PROGRAM P5_04_BatchStatus
VAR
	tonBatchOpen			:TON;
	tPhaseTimeET			:TIME;
	tSubStep1Prod			:TIME;
	tSubStep1				:TIME;
	tSubStep2				:TIME;
	tSubStep3				:TIME;
	tSubStep4				:TIME;
	tSubStep5				:TIME;
	tSubStep6				:TIME;
	tSubStep7				:TIME;
	
	tSubStep1pt				:TIME;
	tSubStep2pt				:TIME;
	tSubStep3pt				:TIME;
	tSubStep4pt				:TIME;
	tSubStep5pt				:TIME;
	tSubStep6pt				:TIME;
	tSubStep7pt				:TIME;
	
	
	bHoldBar1				:BOOL;
	bHoldBar2				:BOOL;
	bHoldBar3				:BOOL;
	bHoldBar4				:BOOL;
	bHoldBar5				:BOOL;
	bHoldBar6				:BOOL;
	bHoldBar7				:BOOL;
	
	
	iCurrProc				:INT;
	

END_VAR
VAR // added by the converter: edge detectors and wires of the graphical bodies
    _w1, _w2, _w3, _w4, _w5, _w6, _w7, _w8, _w9, _w10, _w11, _w12, _w13, _w14, _w15 : TIME;
    _w16 : BOOL;
END_VAR

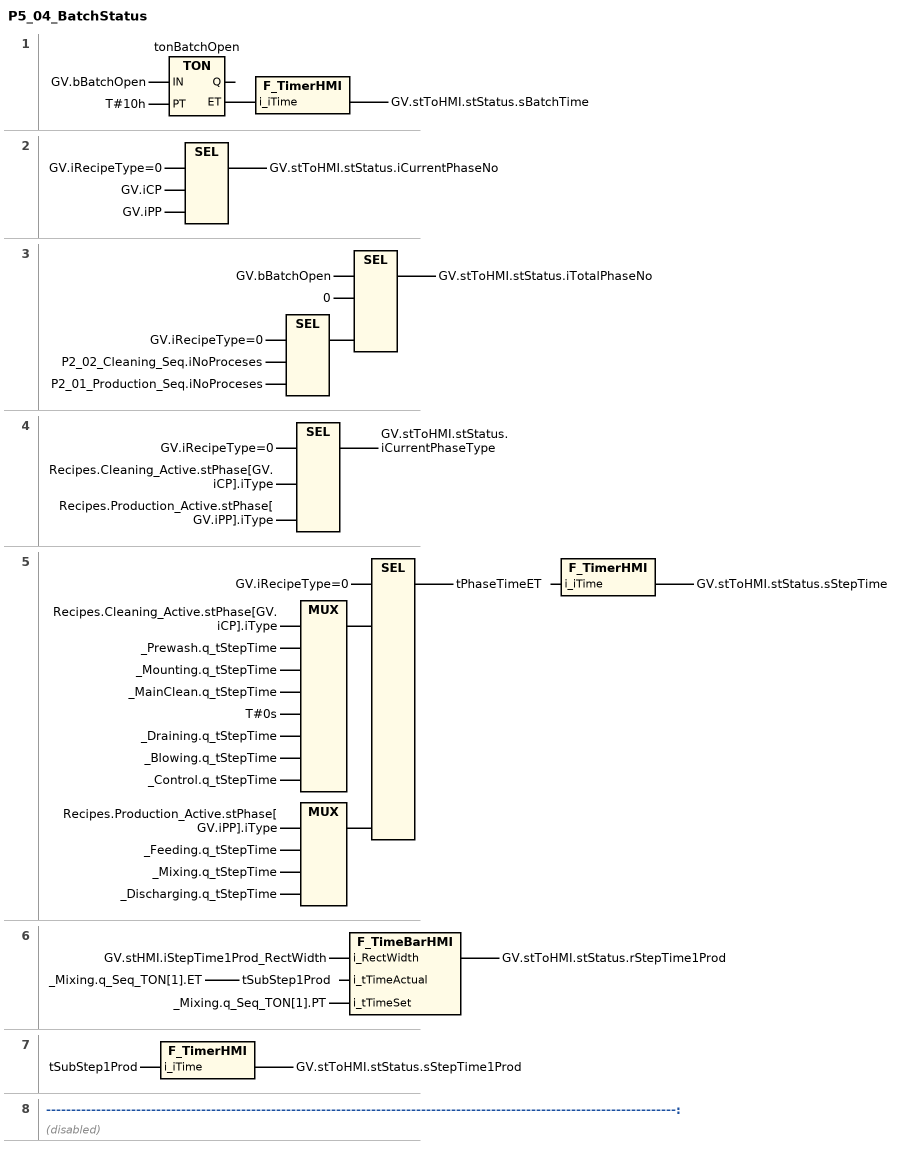
// NETWORK 1
tonBatchOpen(IN := GV.bBatchOpen, PT := T#10h); // TON
GV.stToHMI.stStatus.sBatchTime := F_TimerHMI(i_iTime := tonBatchOpen.ET);

// NETWORK 2
GV.stToHMI.stStatus.iCurrentPhaseNo := SEL(GV.iRecipeType=0, GV.iCP, GV.iPP);

// NETWORK 3
GV.stToHMI.stStatus.iTotalPhaseNo := SEL(GV.bBatchOpen, 0, SEL(GV.iRecipeType=0, P2_02_Cleaning_Seq.iNoProceses, P2_01_Production_Seq.iNoProceses));

// NETWORK 4
GV.stToHMI.stStatus.iCurrentPhaseType := SEL(GV.iRecipeType=0, Recipes.Cleaning_Active.stPhase[GV.iCP].iType, Recipes.Production_Active.stPhase[GV.iPP].iType);

// NETWORK 5
_w1 := SEL(GV.iRecipeType=0, MUX(Recipes.Cleaning_Active.stPhase[GV.iCP].iType, _Prewash.q_tStepTime, _Mounting.q_tStepTime, _MainClean.q_tStepTime, T#0s, _Draining.q_tStepTime, _Blowing.q_tStepTime, _Control.q_tStepTime), MUX(Recipes.Production_Active.stPhase[GV.iPP].iType, _Feeding.q_tStepTime, _Mixing.q_tStepTime, _Discharging.q_tStepTime));
tPhaseTimeET := _w1;
GV.stToHMI.stStatus.sStepTime := F_TimerHMI(i_iTime := _w1);

// NETWORK 6
tSubStep1Prod := _Mixing.q_Seq_TON[1].ET;
GV.stToHMI.stStatus.rStepTime1Prod := F_TimeBarHMI(i_RectWidth := GV.stHMI.iStepTime1Prod_RectWidth, i_tTimeActual := _Mixing.q_Seq_TON[1].ET, i_tTimeSet := _Mixing.q_Seq_TON[1].PT);

// NETWORK 7
GV.stToHMI.stStatus.sStepTime1Prod := F_TimerHMI(i_iTime := tSubStep1Prod);

// NETWORK 8 (disabled)
// label: ------------------------------------------------------------------------------------------------------------------------------

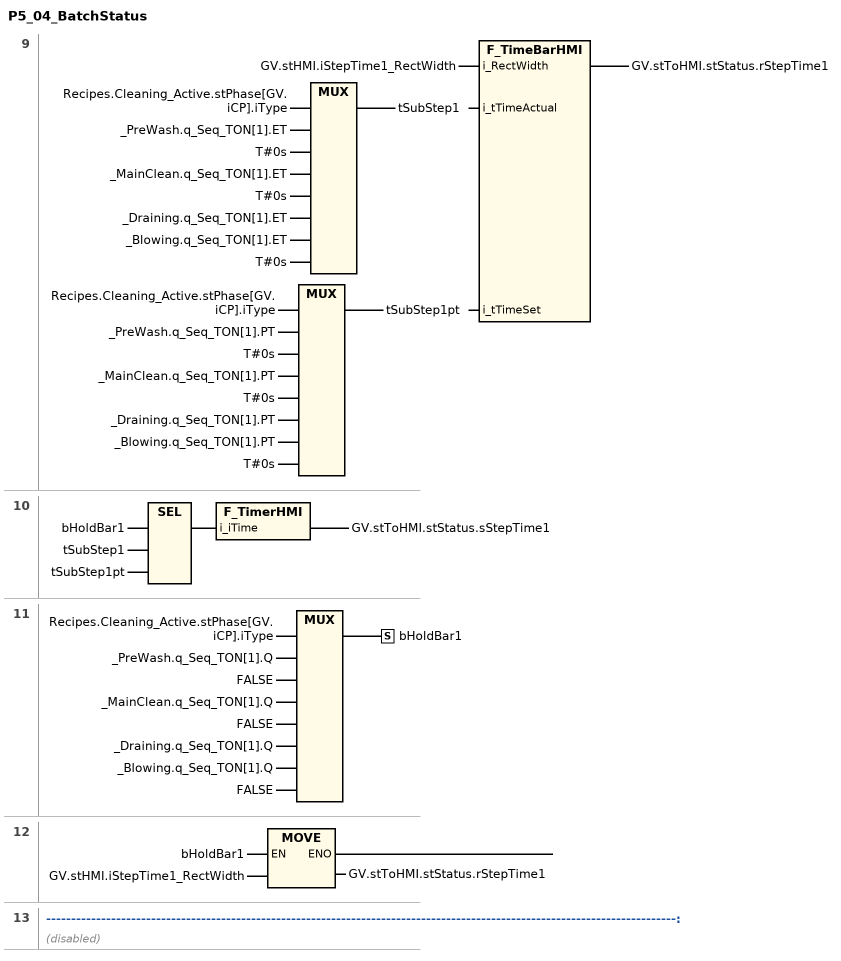
// NETWORK 9
_w2 := MUX(Recipes.Cleaning_Active.stPhase[GV.iCP].iType, _PreWash.q_Seq_TON[1].ET, T#0s, _MainClean.q_Seq_TON[1].ET, T#0s, _Draining.q_Seq_TON[1].ET, _Blowing.q_Seq_TON[1].ET, T#0s);
tSubStep1 := _w2;
_w3 := MUX(Recipes.Cleaning_Active.stPhase[GV.iCP].iType, _PreWash.q_Seq_TON[1].PT, T#0s, _MainClean.q_Seq_TON[1].PT, T#0s, _Draining.q_Seq_TON[1].PT, _Blowing.q_Seq_TON[1].PT, T#0s);
tSubStep1pt := _w3;
GV.stToHMI.stStatus.rStepTime1 := F_TimeBarHMI(i_RectWidth := GV.stHMI.iStepTime1_RectWidth, i_tTimeActual := _w2, i_tTimeSet := _w3);

// NETWORK 10
GV.stToHMI.stStatus.sStepTime1 := F_TimerHMI(i_iTime := SEL(bHoldBar1, tSubStep1, tSubStep1pt));

// NETWORK 11
bHoldBar1 S= MUX(Recipes.Cleaning_Active.stPhase[GV.iCP].iType, _PreWash.q_Seq_TON[1].Q, FALSE, _MainClean.q_Seq_TON[1].Q, FALSE, _Draining.q_Seq_TON[1].Q, _Blowing.q_Seq_TON[1].Q, FALSE);

// NETWORK 12
IF bHoldBar1 THEN GV.stToHMI.stStatus.rStepTime1 := GV.stHMI.iStepTime1_RectWidth; END_IF

// NETWORK 13 (disabled)
// label: ------------------------------------------------------------------------------------------------------------------------------

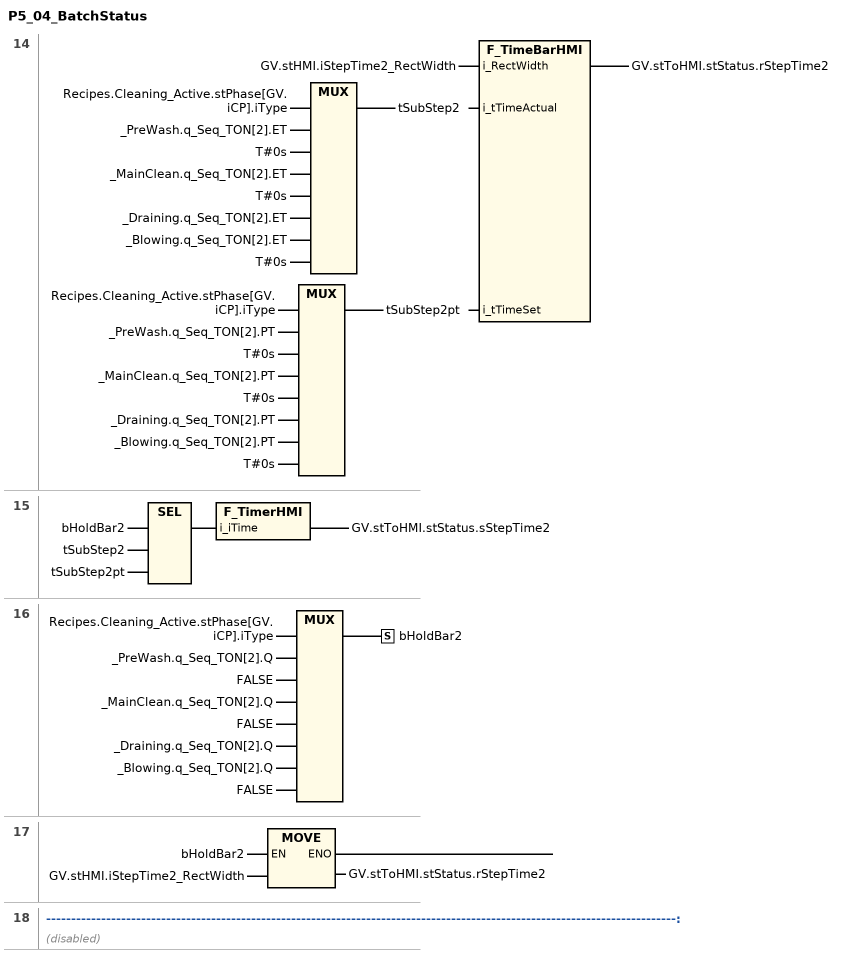
// NETWORK 14
_w4 := MUX(Recipes.Cleaning_Active.stPhase[GV.iCP].iType, _PreWash.q_Seq_TON[2].ET, T#0s, _MainClean.q_Seq_TON[2].ET, T#0s, _Draining.q_Seq_TON[2].ET, _Blowing.q_Seq_TON[2].ET, T#0s);
tSubStep2 := _w4;
_w5 := MUX(Recipes.Cleaning_Active.stPhase[GV.iCP].iType, _PreWash.q_Seq_TON[2].PT, T#0s, _MainClean.q_Seq_TON[2].PT, T#0s, _Draining.q_Seq_TON[2].PT, _Blowing.q_Seq_TON[2].PT, T#0s);
tSubStep2pt := _w5;
GV.stToHMI.stStatus.rStepTime2 := F_TimeBarHMI(i_RectWidth := GV.stHMI.iStepTime2_RectWidth, i_tTimeActual := _w4, i_tTimeSet := _w5);

// NETWORK 15
GV.stToHMI.stStatus.sStepTime2 := F_TimerHMI(i_iTime := SEL(bHoldBar2, tSubStep2, tSubStep2pt));

// NETWORK 16
bHoldBar2 S= MUX(Recipes.Cleaning_Active.stPhase[GV.iCP].iType, _PreWash.q_Seq_TON[2].Q, FALSE, _MainClean.q_Seq_TON[2].Q, FALSE, _Draining.q_Seq_TON[2].Q, _Blowing.q_Seq_TON[2].Q, FALSE);

// NETWORK 17
IF bHoldBar2 THEN GV.stToHMI.stStatus.rStepTime2 := GV.stHMI.iStepTime2_RectWidth; END_IF

// NETWORK 18 (disabled)
// label: ------------------------------------------------------------------------------------------------------------------------------

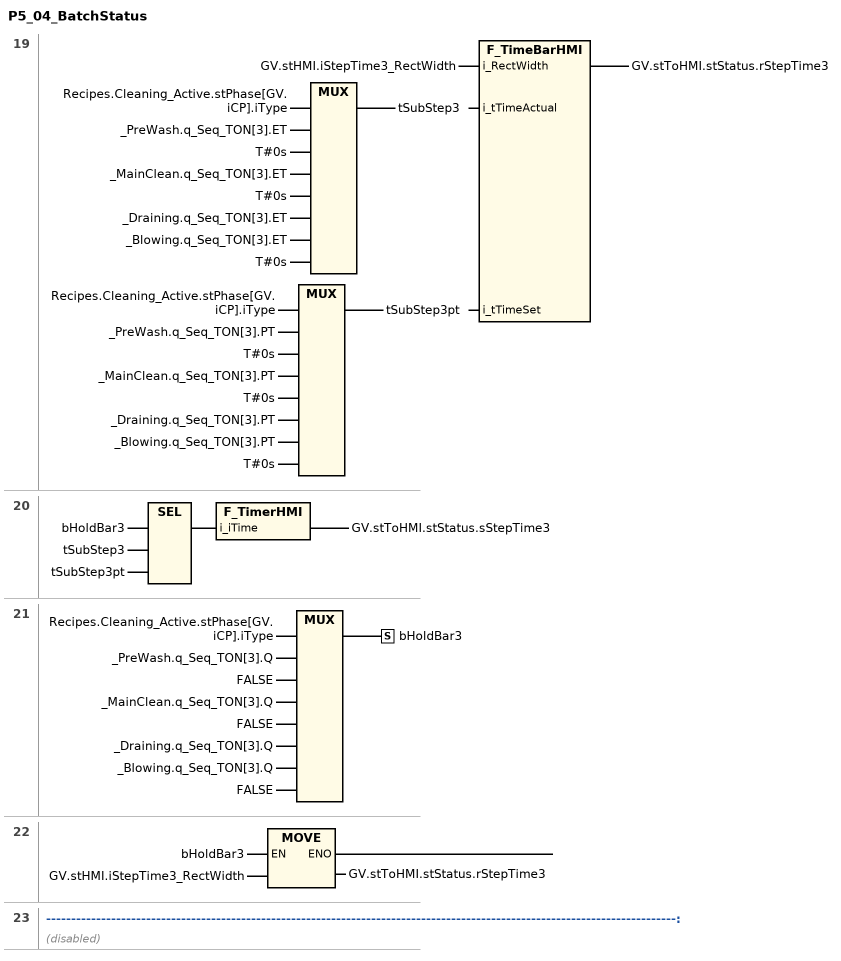
// NETWORK 19
_w6 := MUX(Recipes.Cleaning_Active.stPhase[GV.iCP].iType, _PreWash.q_Seq_TON[3].ET, T#0s, _MainClean.q_Seq_TON[3].ET, T#0s, _Draining.q_Seq_TON[3].ET, _Blowing.q_Seq_TON[3].ET, T#0s);
tSubStep3 := _w6;
_w7 := MUX(Recipes.Cleaning_Active.stPhase[GV.iCP].iType, _PreWash.q_Seq_TON[3].PT, T#0s, _MainClean.q_Seq_TON[3].PT, T#0s, _Draining.q_Seq_TON[3].PT, _Blowing.q_Seq_TON[3].PT, T#0s);
tSubStep3pt := _w7;
GV.stToHMI.stStatus.rStepTime3 := F_TimeBarHMI(i_RectWidth := GV.stHMI.iStepTime3_RectWidth, i_tTimeActual := _w6, i_tTimeSet := _w7);

// NETWORK 20
GV.stToHMI.stStatus.sStepTime3 := F_TimerHMI(i_iTime := SEL(bHoldBar3, tSubStep3, tSubStep3pt));

// NETWORK 21
bHoldBar3 S= MUX(Recipes.Cleaning_Active.stPhase[GV.iCP].iType, _PreWash.q_Seq_TON[3].Q, FALSE, _MainClean.q_Seq_TON[3].Q, FALSE, _Draining.q_Seq_TON[3].Q, _Blowing.q_Seq_TON[3].Q, FALSE);

// NETWORK 22
IF bHoldBar3 THEN GV.stToHMI.stStatus.rStepTime3 := GV.stHMI.iStepTime3_RectWidth; END_IF

// NETWORK 23 (disabled)
// label: ------------------------------------------------------------------------------------------------------------------------------

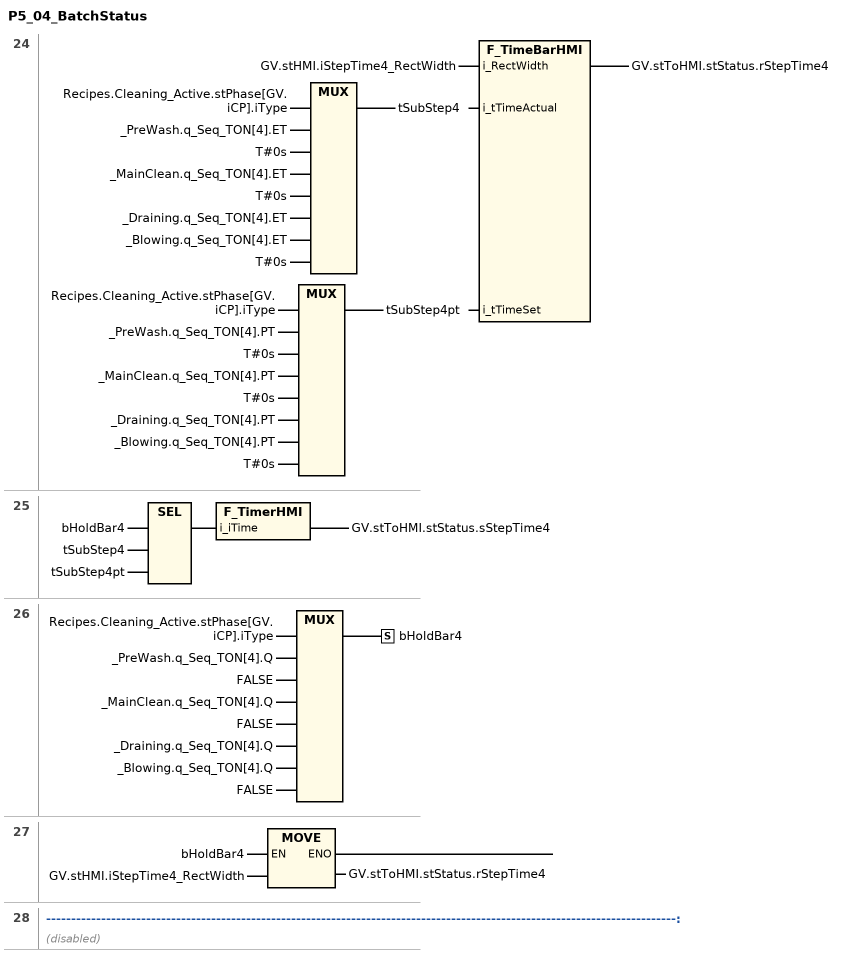
// NETWORK 24
_w8 := MUX(Recipes.Cleaning_Active.stPhase[GV.iCP].iType, _PreWash.q_Seq_TON[4].ET, T#0s, _MainClean.q_Seq_TON[4].ET, T#0s, _Draining.q_Seq_TON[4].ET, _Blowing.q_Seq_TON[4].ET, T#0s);
tSubStep4 := _w8;
_w9 := MUX(Recipes.Cleaning_Active.stPhase[GV.iCP].iType, _PreWash.q_Seq_TON[4].PT, T#0s, _MainClean.q_Seq_TON[4].PT, T#0s, _Draining.q_Seq_TON[4].PT, _Blowing.q_Seq_TON[4].PT, T#0s);
tSubStep4pt := _w9;
GV.stToHMI.stStatus.rStepTime4 := F_TimeBarHMI(i_RectWidth := GV.stHMI.iStepTime4_RectWidth, i_tTimeActual := _w8, i_tTimeSet := _w9);

// NETWORK 25
GV.stToHMI.stStatus.sStepTime4 := F_TimerHMI(i_iTime := SEL(bHoldBar4, tSubStep4, tSubStep4pt));

// NETWORK 26
bHoldBar4 S= MUX(Recipes.Cleaning_Active.stPhase[GV.iCP].iType, _PreWash.q_Seq_TON[4].Q, FALSE, _MainClean.q_Seq_TON[4].Q, FALSE, _Draining.q_Seq_TON[4].Q, _Blowing.q_Seq_TON[4].Q, FALSE);

// NETWORK 27
IF bHoldBar4 THEN GV.stToHMI.stStatus.rStepTime4 := GV.stHMI.iStepTime4_RectWidth; END_IF

// NETWORK 28 (disabled)
// label: ------------------------------------------------------------------------------------------------------------------------------

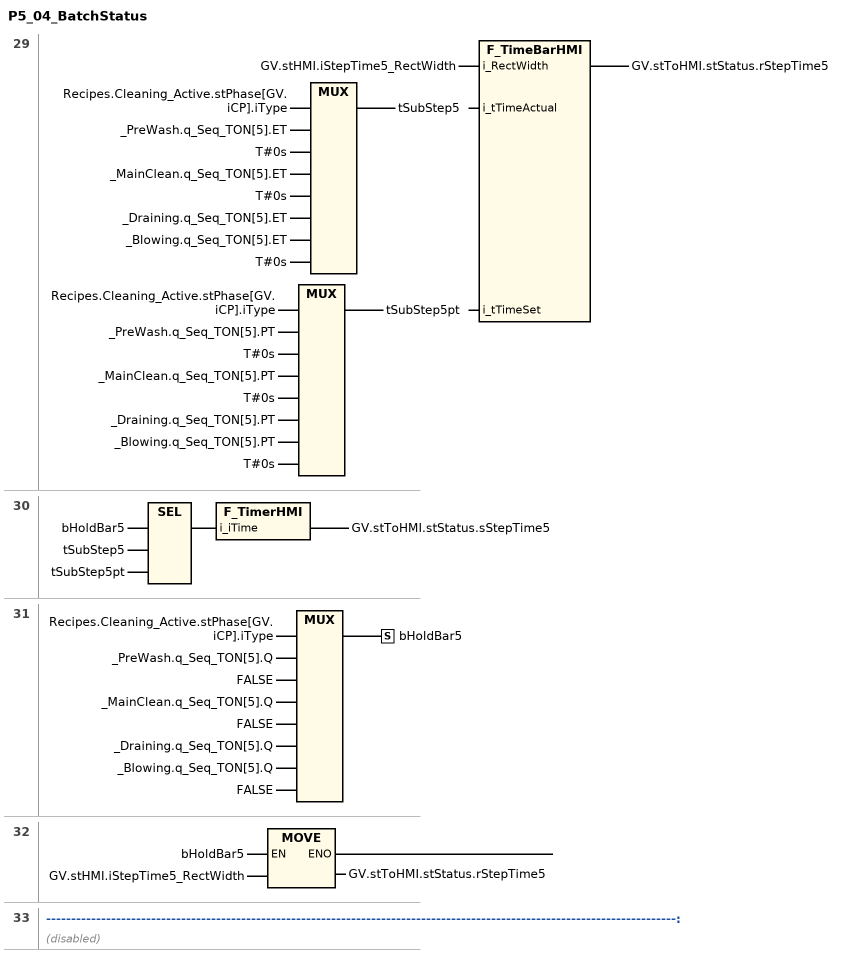
// NETWORK 29
_w10 := MUX(Recipes.Cleaning_Active.stPhase[GV.iCP].iType, _PreWash.q_Seq_TON[5].ET, T#0s, _MainClean.q_Seq_TON[5].ET, T#0s, _Draining.q_Seq_TON[5].ET, _Blowing.q_Seq_TON[5].ET, T#0s);
tSubStep5 := _w10;
_w11 := MUX(Recipes.Cleaning_Active.stPhase[GV.iCP].iType, _PreWash.q_Seq_TON[5].PT, T#0s, _MainClean.q_Seq_TON[5].PT, T#0s, _Draining.q_Seq_TON[5].PT, _Blowing.q_Seq_TON[5].PT, T#0s);
tSubStep5pt := _w11;
GV.stToHMI.stStatus.rStepTime5 := F_TimeBarHMI(i_RectWidth := GV.stHMI.iStepTime5_RectWidth, i_tTimeActual := _w10, i_tTimeSet := _w11);

// NETWORK 30
GV.stToHMI.stStatus.sStepTime5 := F_TimerHMI(i_iTime := SEL(bHoldBar5, tSubStep5, tSubStep5pt));

// NETWORK 31
bHoldBar5 S= MUX(Recipes.Cleaning_Active.stPhase[GV.iCP].iType, _PreWash.q_Seq_TON[5].Q, FALSE, _MainClean.q_Seq_TON[5].Q, FALSE, _Draining.q_Seq_TON[5].Q, _Blowing.q_Seq_TON[5].Q, FALSE);

// NETWORK 32
IF bHoldBar5 THEN GV.stToHMI.stStatus.rStepTime5 := GV.stHMI.iStepTime5_RectWidth; END_IF

// NETWORK 33 (disabled)
// label: ------------------------------------------------------------------------------------------------------------------------------

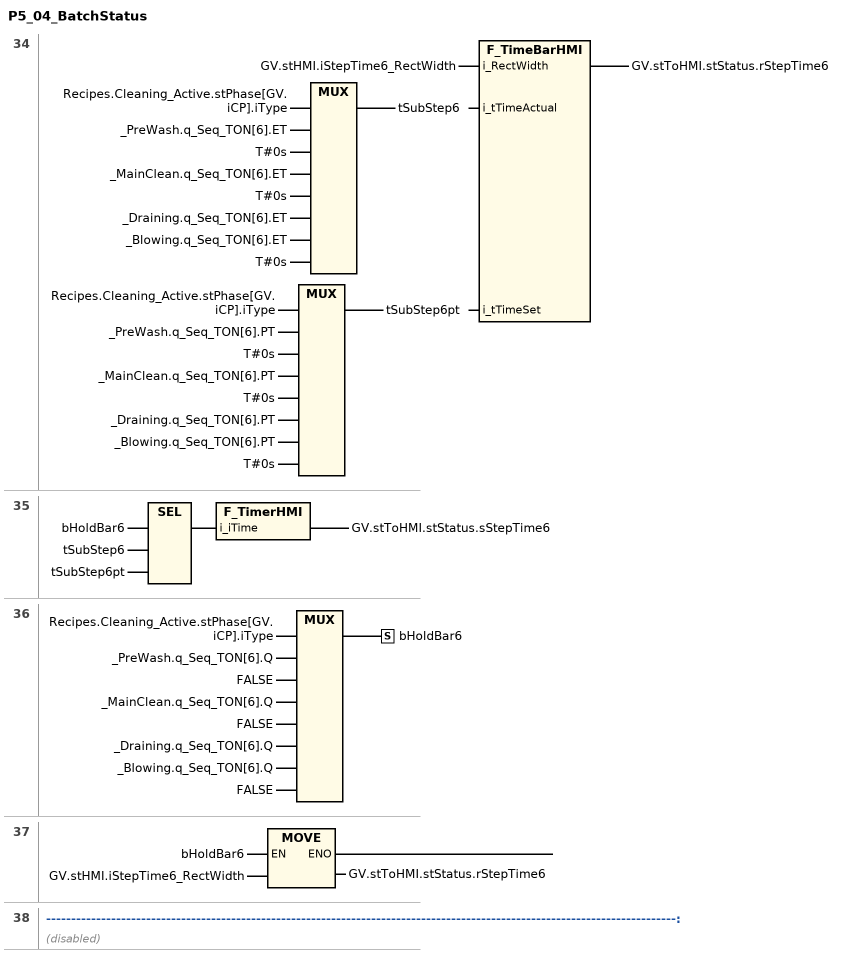
// NETWORK 34
_w12 := MUX(Recipes.Cleaning_Active.stPhase[GV.iCP].iType, _PreWash.q_Seq_TON[6].ET, T#0s, _MainClean.q_Seq_TON[6].ET, T#0s, _Draining.q_Seq_TON[6].ET, _Blowing.q_Seq_TON[6].ET, T#0s);
tSubStep6 := _w12;
_w13 := MUX(Recipes.Cleaning_Active.stPhase[GV.iCP].iType, _PreWash.q_Seq_TON[6].PT, T#0s, _MainClean.q_Seq_TON[6].PT, T#0s, _Draining.q_Seq_TON[6].PT, _Blowing.q_Seq_TON[6].PT, T#0s);
tSubStep6pt := _w13;
GV.stToHMI.stStatus.rStepTime6 := F_TimeBarHMI(i_RectWidth := GV.stHMI.iStepTime6_RectWidth, i_tTimeActual := _w12, i_tTimeSet := _w13);

// NETWORK 35
GV.stToHMI.stStatus.sStepTime6 := F_TimerHMI(i_iTime := SEL(bHoldBar6, tSubStep6, tSubStep6pt));

// NETWORK 36
bHoldBar6 S= MUX(Recipes.Cleaning_Active.stPhase[GV.iCP].iType, _PreWash.q_Seq_TON[6].Q, FALSE, _MainClean.q_Seq_TON[6].Q, FALSE, _Draining.q_Seq_TON[6].Q, _Blowing.q_Seq_TON[6].Q, FALSE);

// NETWORK 37
IF bHoldBar6 THEN GV.stToHMI.stStatus.rStepTime6 := GV.stHMI.iStepTime6_RectWidth; END_IF

// NETWORK 38 (disabled)
// label: ------------------------------------------------------------------------------------------------------------------------------

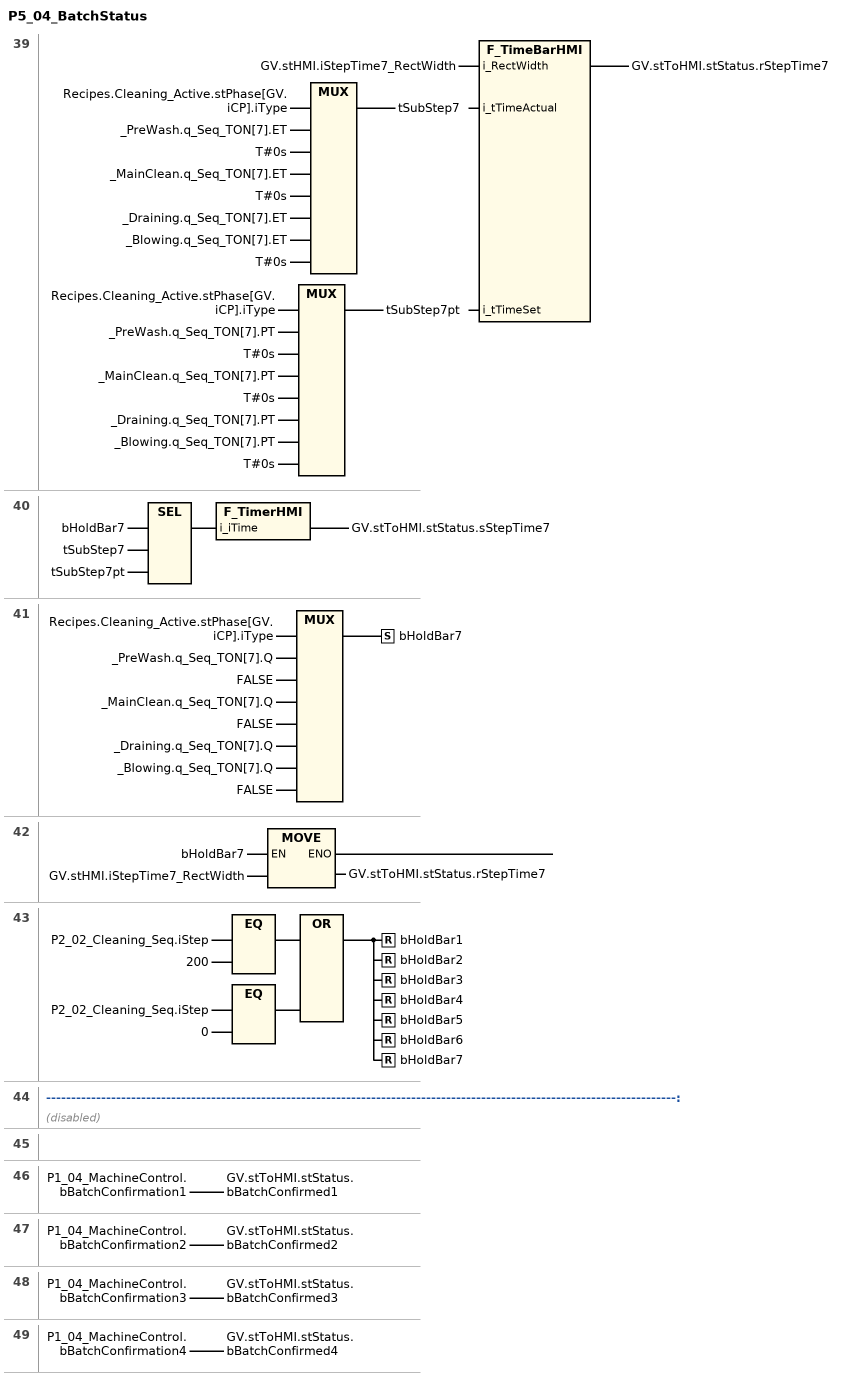
// NETWORK 39
_w14 := MUX(Recipes.Cleaning_Active.stPhase[GV.iCP].iType, _PreWash.q_Seq_TON[7].ET, T#0s, _MainClean.q_Seq_TON[7].ET, T#0s, _Draining.q_Seq_TON[7].ET, _Blowing.q_Seq_TON[7].ET, T#0s);
tSubStep7 := _w14;
_w15 := MUX(Recipes.Cleaning_Active.stPhase[GV.iCP].iType, _PreWash.q_Seq_TON[7].PT, T#0s, _MainClean.q_Seq_TON[7].PT, T#0s, _Draining.q_Seq_TON[7].PT, _Blowing.q_Seq_TON[7].PT, T#0s);
tSubStep7pt := _w15;
GV.stToHMI.stStatus.rStepTime7 := F_TimeBarHMI(i_RectWidth := GV.stHMI.iStepTime7_RectWidth, i_tTimeActual := _w14, i_tTimeSet := _w15);

// NETWORK 40
GV.stToHMI.stStatus.sStepTime7 := F_TimerHMI(i_iTime := SEL(bHoldBar7, tSubStep7, tSubStep7pt));

// NETWORK 41
bHoldBar7 S= MUX(Recipes.Cleaning_Active.stPhase[GV.iCP].iType, _PreWash.q_Seq_TON[7].Q, FALSE, _MainClean.q_Seq_TON[7].Q, FALSE, _Draining.q_Seq_TON[7].Q, _Blowing.q_Seq_TON[7].Q, FALSE);

// NETWORK 42
IF bHoldBar7 THEN GV.stToHMI.stStatus.rStepTime7 := GV.stHMI.iStepTime7_RectWidth; END_IF

// NETWORK 43
_w16 := P2_02_Cleaning_Seq.iStep = 200 OR P2_02_Cleaning_Seq.iStep = 0;
bHoldBar1 R= _w16;
bHoldBar2 R= _w16;
bHoldBar3 R= _w16;
bHoldBar4 R= _w16;
bHoldBar5 R= _w16;
bHoldBar6 R= _w16;
bHoldBar7 R= _w16;

// NETWORK 44 (disabled)
// label: ------------------------------------------------------------------------------------------------------------------------------

// NETWORK 45

// NETWORK 46
GV.stToHMI.stStatus.bBatchConfirmed1 := P1_04_MachineControl.bBatchConfirmation1;

// NETWORK 47
GV.stToHMI.stStatus.bBatchConfirmed2 := P1_04_MachineControl.bBatchConfirmation2;

// NETWORK 48
GV.stToHMI.stStatus.bBatchConfirmed3 := P1_04_MachineControl.bBatchConfirmation3;

// NETWORK 49
GV.stToHMI.stStatus.bBatchConfirmed4 := P1_04_MachineControl.bBatchConfirmation4;

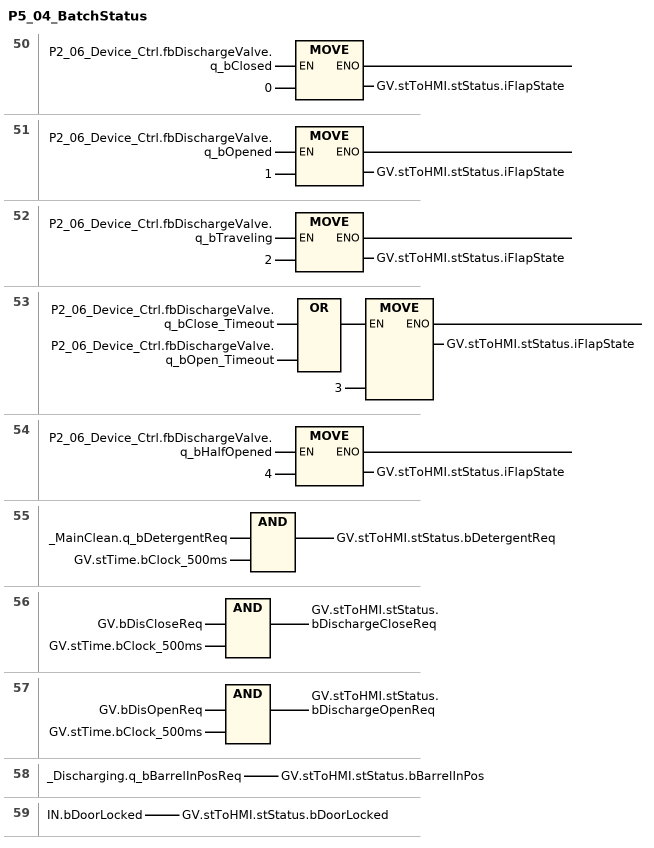
// NETWORK 50
IF P2_06_Device_Ctrl.fbDischargeValve.q_bClosed THEN GV.stToHMI.stStatus.iFlapState := 0; END_IF

// NETWORK 51
IF P2_06_Device_Ctrl.fbDischargeValve.q_bOpened THEN GV.stToHMI.stStatus.iFlapState := 1; END_IF

// NETWORK 52
IF P2_06_Device_Ctrl.fbDischargeValve.q_bTraveling THEN GV.stToHMI.stStatus.iFlapState := 2; END_IF

// NETWORK 53
IF P2_06_Device_Ctrl.fbDischargeValve.q_bClose_Timeout OR P2_06_Device_Ctrl.fbDischargeValve.q_bOpen_Timeout THEN
    GV.stToHMI.stStatus.iFlapState := 3;
END_IF

// NETWORK 54
IF P2_06_Device_Ctrl.fbDischargeValve.q_bHalfOpened THEN GV.stToHMI.stStatus.iFlapState := 4; END_IF

// NETWORK 55
GV.stToHMI.stStatus.bDetergentReq := _MainClean.q_bDetergentReq AND GV.stTime.bClock_500ms;

// NETWORK 56
GV.stToHMI.stStatus.bDischargeCloseReq := GV.bDisCloseReq AND GV.stTime.bClock_500ms;

// NETWORK 57
GV.stToHMI.stStatus.bDischargeOpenReq := GV.bDisOpenReq AND GV.stTime.bClock_500ms;

// NETWORK 58
GV.stToHMI.stStatus.bBarrelInPos := _Discharging.q_bBarrelInPosReq;

// NETWORK 59
GV.stToHMI.stStatus.bDoorLocked := IN.bDoorLocked;

END_PROGRAM

(* stored: Version 1.1.0.1
   POU P5_04_BatchStatus: Id {20236771-a5db-4126-ae7f-014e653563e0}, SpecialFunc None *)
